{attribute 'GeneratedUsingTerminal: EL9400--0000'}
{attribute addProperty BoxType "EL9400--0000"}
{attribute addProperty Description "EL9400 E-Bus Power Supplier"}
{attribute addProperty Physics "KK"}
{attribute addProperty Id "EL9400"}
{attribute addProperty CRC "132600645"}
{attribute addProperty Size "0"}
TYPE EL9400_07E75345 EXTENDS EtcSlaveTerminalBase_947E5A46 :
STRUCT
END_STRUCT
END_TYPE

(* stored: Version 1.2.0.0, ProductVersion 3.1.4024.11
   DUT EL9400_07E75345: Id {4cd87ecb-459a-4aaa-b64c-3165cd9ccb18} *)
